(* PLC project Unnamed, Unknown Unnamed 1 *)
(* stored: creationDateTime 2024-12-02T16:53:49, modificationDateTime 2024-12-02T17:14:04 *)

PROGRAM exp1
  VAR_INPUT
    Start : BOOL;
  END_VAR
  VAR_OUTPUT
    Lamp : BOOL;
  END_VAR

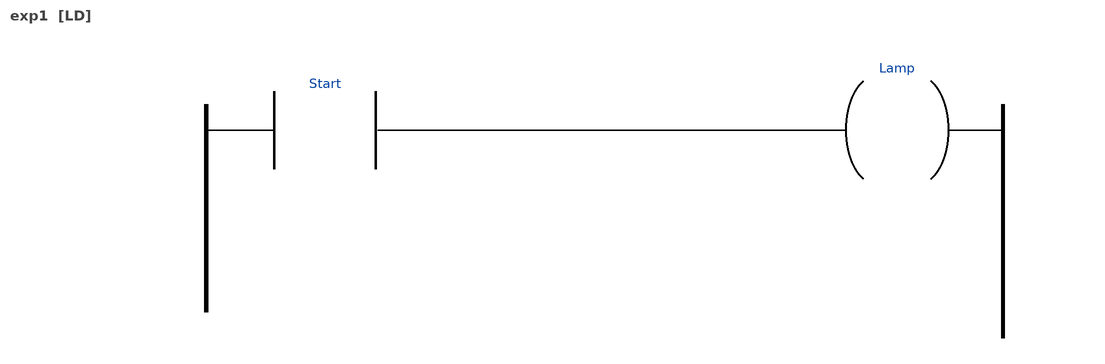
(* LD diagram, written out as Structured Text *)
Lamp := Start;
END_PROGRAM

CONFIGURATION Config0
  RESOURCE Res0 ON PLC
    TASK task0(INTERVAL := T#20ms, PRIORITY := 0);
    PROGRAM instance0 WITH task0 : exp1;
  END_RESOURCE
END_CONFIGURATION
